TYPE (* A Structured Data Type *)
  (* Standard: 61499-2 *)
  (* Version 0.1, 2003-12-05, JHC, Rockwell Automation, Renamed from NEWSTRUCT. *)
  (* Version 0.0, 2000-05-27, JHC, Rockwell Automation *)
  (* Compiler header: package fb.rt.cs725; *)
  (* ASN.1 tag PRIVATE 5 *)
  BagDetail : STRUCT
    bagYValue : DINT;
    bagXValue : DINT;
    conId : DINT;
  END_STRUCT;
END_TYPE
